ABB RobotStudio station: proyecto_CI.rsstn

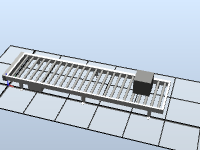
Station proyecto_CI (saved by RobotStudio 6.6.7701.1025)
Layout (positions relative to the parent item):
  - 1200_4800_h2 [part, from Equipment\Conveyor 1200 4800 h2.rslib]
  - Componente inteligente_2 [smart component]
      signals: DI on, DI nuevo, DO holi, DO sen, DI ok
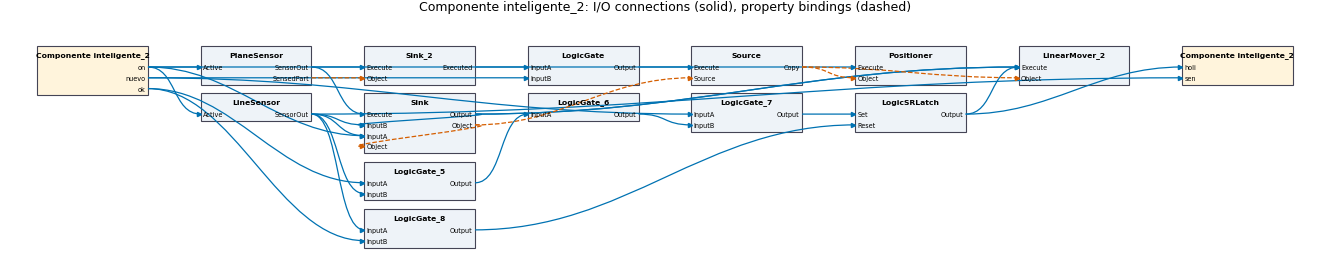
      connections:
        PlaneSensor.SensorOut -> Sink.Execute
        PlaneSensor.SensorOut -> Sink_2.Execute
        Componente inteligente_2.on -> PlaneSensor.Active
        Componente inteligente_2.on -> Positioner.Execute
        Sink_2.Executed -> LogicGate.InputA
        Componente inteligente_2.nuevo -> LogicGate.InputB
        LogicGate.Output -> Source.Execute
        Componente inteligente_2.on -> LineSensor.Active
        LineSensor.SensorOut -> LogicGate_2.InputB
        LogicGate_2.Output -> LinearMover_2.Execute
        LineSensor.SensorOut -> LogicGate_3.InputA
        LogicGate_3.Output -> LogicGate_4.InputB
        Componente inteligente_2.on -> LogicGate_4.InputA
        LogicGate_4.Output -> LinearMover_2.Execute
        LogicSRLatch.Output -> LinearMover_2.Execute
        LogicSRLatch.Output -> Componente inteligente_2.holi
        LineSensor.SensorOut -> Componente inteligente_2.sen
        Componente inteligente_2.ok -> LogicGate_5.InputA
        LineSensor.SensorOut -> LogicGate_5.InputB
        LogicGate_5.Output -> LogicGate_6.InputA
        Componente inteligente_2.nuevo -> LogicGate_7.InputA
        LogicGate_6.Output -> LogicGate_7.InputB
        LogicGate_7.Output -> LogicSRLatch.Set
        LogicGate_8.Output -> LogicSRLatch.Reset
        LineSensor.SensorOut -> LogicGate_8.InputA
        Componente inteligente_2.ok -> LogicGate_8.InputB
        LinearMover.Object => Sink.Object
        LinearMover.Object => Source.Source
        Source.Copy => LinearMover_2.Object
        PlaneSensor.SensedPart => Sink_2.Object
        Source.Copy => Positioner.Object
    - PlaneSensor [smart component, from Components\PlaneSensor.rslib]
        properties: Origin=[5 0 0]; Axis1=[0 0 1]; Axis2=[0 1 0]; SensedPart=(none)
      - _sensorPart_ [part]
    - Source [smart component, from Components\Source.rslib]
        properties: Source=Pieza_2; Copy=Pieza_2_152; Parent=(none); Position=[0 0 0]; Orientation=[0 0 0]; Transient=false; PhysicsBehavior=0
    - Sink_2 [smart component, from Components\Sink.rslib]
        properties: Object=(none)
    - LinearMover_2 [smart component, from Components\LinearMover.rslib]
        properties: Object=Pieza_2_152; Direction=[1 0 0]; Speed=1; Reference=Global; ReferenceObject=(none)
    - Positioner [smart component, from Components\Positioner.rslib]
        properties: Object=Pieza_2_152; Position=[0 0 0]; Orientation=[0 0 0]; Reference=Global; ReferenceObject=(none)
    - LogicGate [smart component, from Components\LogicGate.rslib]
        properties: Operator=OR; Delay=0
    - LineSensor [smart component, from Components\LineSensor.rslib]
        properties: Start=[2.386925 0.626637 0.450736]; End=[2.386925 0.626637 0.493736]; Radius=0.01; SensedPart=(none); SensedPoint=[0 0 0]
      - _sensorPart_ [part]
    - LogicSRLatch [smart component, from Components\LogicSRLatch.rslib]
    - LogicGate_5 [smart component, from Components\LogicGate.rslib]
        properties: Operator=XOR; Delay=0
    - LogicGate_6 [smart component, from Components\LogicGate.rslib]
        properties: Operator=NOT; Delay=0
    - LogicGate_7 [smart component, from Components\LogicGate.rslib]
        properties: Operator=OR; Delay=0
    - LogicGate_8 [smart component, from Components\LogicGate.rslib]
        properties: Operator=XOR; Delay=0
  - Pieza_2 [part]
  - Pieza_2_152 [part] at (3936, 0, 0) mm
